# EPICS autosave request: apps/plcApp/Db/torus_LHe_settings.req
#
# torus_LHe_settings.req - autosave, Torus Helium Alarms
#
# Author: Wesley Moore (wmoore@jlab.org)
# Date:   June 2016
#
# Helium
#
# Cernox
file "torus_ccm_cernox.req"  P=$(P), R=$(R), CCM=A
file "torus_ccm_cernox.req"  P=$(P), R=$(R), CCM=B
file "torus_ccm_cernox.req"  P=$(P), R=$(R), CCM=C
file "torus_ccm_cernox.req"  P=$(P), R=$(R), CCM=D
file "torus_ccm_cernox.req"  P=$(P), R=$(R), CCM=E
file "torus_ccm_cernox.req"  P=$(P), R=$(R), CCM=F
